KUKA KRL program: LeafDataAut3.src, LeafDataAut3.dat

--- LeafDataAut3.src ---
&ACCESS RV
&REL 4
DEFFCT ST_Dim3 LeafDataAut3(eElement:IN,iElement:IN)
   ;FOLD DECL
      DECL Data_LeafAut3 eElement
      DECL INT iElement
      DECL ST_Dim3 stData

      DECL ST_Dim3 stScrew[10],stPocket[3]
      DECL ST_Dim3 stScrewTemp,stPocketTemp
      DECL ST_Dim3 stHandle,stHandleTemp,stKey,stKeyTemp
      DECL INT iScrew,iPocket
   ;ENDFOLD

   SWITCH eElement
      CASE #Screw
         stData = GetScrewPlace(iElement)
      CASE #Pocket
         stData = GetPocketPlace(iElement)
      CASE #PocketDim
         stData = GetPocketDim(iElement)
      DEFAULT
         HALT
   ENDSWITCH

   RETURN stData

ENDFCT

DEFFCT ST_Dim3 GetScrewPlace(iScrew:IN)
   ;FOLD DECL
      DECL INT iScrew
      DECL E_ProfileType eProfileType
      DECL REAL rScrewRefX,rScrewY
      DECL ST_Dim3 stScrew
   ;ENDFOLD (DECL)

   ;ProcessData
   eProfileType = gstProcessData.eProfileType

   ;rScrewRefX,rScrewY
   SWITCH eProfileType
      CASE #Leaf75
         rScrewRefX = rPlateRefDist_Leaf75
         rScrewY = rPlateY_Leaf75
      CASE #Leaf90
         rScrewRefX = rPlateRefDist_Leaf90
         rScrewY = rPlateY_Leaf90
      DEFAULT
         HALT
   ENDSWITCH

   ;stScrew
   stScrew.rX = rScrewRefX + rScrewDist[iScrew]
   stScrew.rY = rScrewY

   ;Return screw data
   RETURN stScrew

ENDFCT

DEFFCT ST_Dim3 GetPocketPlace(iPocket:IN)
   ;FOLD DECL
      DECL INT iPocket
      DECL E_ProfileType eProfileType
      DECL REAL rPocketRefX,rPocketY
      DECL ST_Dim3 stScrew
   ;ENDFOLD (DECL)

   ;ProcessData
   eProfileType = gstProcessData.eProfileType

   ;rPocketRefX,rPocketY
   SWITCH eProfileType
      CASE #Leaf75
         rPocketRefX = rPlateRefDist_Leaf75
         rPocketY = rPlateY_Leaf75
      CASE #Leaf90
         rPocketRefX = rPlateRefDist_Leaf90
         rPocketY = rPlateY_Leaf90
      DEFAULT
         HALT
   ENDSWITCH

   ;stScrew
   stScrew.rX = rPocketRefX + rPocketDist[iPocket]
   stScrew.rY = rPocketY

   ;Return screw data
   RETURN stScrew

ENDFCT

DEFFCT ST_Dim3 GetPocketDim(iPocket:IN)
   ;FOLD DECL
      DECL INT iPocket
      DECL ST_Dim3 stPocketDim
   ;ENDFOLD (DECL)

   ;stPocketDim
   SWITCH iPocket
      CASE 1,3
         stPocketDim = stAuxPocketDim
      CASE 2
         stPocketDim = stMainPocketDim
      DEFAULT
         HALT
   ENDSWITCH

   ;Return pocket dimensions
   RETURN stPocketDim

ENDFCT

--- LeafDataAut3.dat ---
&ACCESS RV
&REL 4
DEFDAT LeafDataAut3 PUBLIC

   GLOBAL ENUM Data_LeafAut3 Screw,Pocket,PocketDim

   ;Reference distance
   DECL CONST REAL rPlateRefDist_Leaf75 = 147.5
   DECL CONST REAL rPlateRefDist_Leaf90 = 152.5

   ;Screw Y coordinate
   DECL CONST REAL rPlateY_Leaf75 = 52.6
   DECL CONST REAL rPlateY_Leaf90 = 67.0

   ;Screws distance
   DECL CONST REAL rScrewDist[10]
   rScrewDist[1]  =   0.0
   rScrewDist[2]  =  195.0
   rScrewDist[3]  =  274.0
   rScrewDist[4]  =  392.0
   rScrewDist[5]  =  543.5
   rScrewDist[6]  =  694.0
   rScrewDist[7]  =  958.0
   rScrewDist[8]  = 1208.0
   rScrewDist[9]  = 1489.5
   rScrewDist[10] = 1685.0

   ;Pocket dimensions
   DECL CONST ST_Dim3 stAuxPocketDim  = {rX 130.0,rY 18.0}
   DECL CONST ST_Dim3 stMainPocketDim = {rX 230.0,rY 18.0}

   ;Pockets distance
   DECL CONST REAL rPocketDist[3]
   rPocketDist[1] =   97.5
   rPocketDist[2] =  826.5
   rPocketDist[3] = 1587.5

ENDDAT
